(* IEC 61131-3 sources: AXOpen/src/data/tests/AXOpen.Repository.Integration.Tests_L4/ax/src, 6 files *)

(* ---- AxoDataExchange.st ---- *)
USING AXOpen.Core;
USING AXOpen;
using AXOpen.Data;

NAMESPACE Exchange_Test_L4

    {S7.extern=ReadWrite}
    CLASS PUBLIC Context EXTENDS AXOpen.Core.AxoContext
        VAR PUBLIC

            DataManager  : ProcessManager;

        END_VAR

        METHOD OVERRIDE Main

        END_METHOD
    END_CLASS

    {S7.extern=ReadWrite}
    CLASS PUBLIC ProcessManager EXTENDS AXOpen.Data.AxoDataExchange
        VAR PUBLIC
            {#ix-generic:TOnline}
            {#ix-generic:TPlain as POCO}
            {#ix-attr:[AXOpen.Data.AxoDataEntityAttribute]}
            Set : ProcessData;
        END_VAR
    END_CLASS

    {S7.extern=ReadWrite}
    CLASS PUBLIC ProcessData EXTENDS AXOpen.Data.AxoDataEntity
        VAR PUBLIC
            vString : STRING;
            vInt : INT;
            vBool : BOOL;
            NestObj : NestedObject;
        END_VAR
    END_CLASS

    {S7.extern=ReadWrite}
    CLASS PUBLIC NestedObject
        VAR PUBLIC
            vString : STRING;
            vInt : INT;
            vBool : BOOL;
        END_VAR
    END_CLASS

END_NAMESPACE

(* ---- AxoDataExchange_Test_L4.st ---- *)
USING AXOpen.Core;
USING AXOpen;
using AXOpen.Data;

NAMESPACE DataFramentsExchange_Test_L4

    //<ContextDeclaration>
    {S7.extern=ReadWrite}
    CLASS PUBLIC Context EXTENDS AXOpen.Core.AxoContext
        VAR PUBLIC

            DataManager  : AxoProcessDataManager_Test_L4;

        END_VAR

        METHOD OVERRIDE Main

        END_METHOD
    END_CLASS
    //</ContextDeclaration>

    //<AxoProcessDataManagerDeclaration>
    {S7.extern=ReadWrite}
    CLASS PUBLIC AxoProcessDataManager_Test_L4 EXTENDS AXOpen.Data.AxoDataExchange
        VAR PUBLIC
            {#ix-generic:TOnline}
            {#ix-generic:TPlain as POCO}
            {#ix-attr:[AXOpen.Data.AxoDataEntityAttribute]}
            Set : AxoProcessData_Test_L4; // <- Manager will operate on this member.
        END_VAR
    END_CLASS
    //</AxoProcessDataManagerDeclaration>

    //<AxoProcessDataDeclaration>
    {S7.extern=ReadWrite}
    CLASS PUBLIC AxoProcessData_Test_L4 EXTENDS AXOpen.Data.AxoDataEntity
        VAR PUBLIC
            vString : STRING;
            vInt : INT;
            vBool : BOOL;
            NestObj : NestingData;
        END_VAR
    END_CLASS
    //</AxoProcessDataDeclaration>

    {S7.extern=ReadWrite}
    CLASS PUBLIC NestingData
        VAR PUBLIC
            vString : STRING;
            vInt : INT;
            vBool : BOOL;
        END_VAR
    END_CLASS

END_NAMESPACE

(* ---- AxoDataFragmentExchange.st ---- *)
USING AXOpen.Core;
USING AXOpen.Data;

NAMESPACE FragmentExchange_Test_L4

    {S7.extern=ReadWrite}
    CLASS PUBLIC Context EXTENDS AXOpen.Core.AxoContext
        VAR PUBLIC
            DataManager  : FragmentProcessDataManager;
        END_VAR

        METHOD OVERRIDE Main

        END_METHOD
    END_CLASS

    {S7.extern=ReadWrite}
    CLASS PUBLIC FragmentProcessDataManager
        EXTENDS AXOpen.Data.AxoDataFragmentExchange
        VAR PUBLIC
            {#ix-attr:[AXOpen.Data.AxoDataFragmentAttribute]}
            Header : HeaderManager;

            {#ix-attr:[AXOpen.Data.AxoDataFragmentAttribute]}
            St1 : StationManager;

        END_VAR
    END_CLASS

    {S7.extern=ReadWrite}
    CLASS PUBLIC HeaderManager
        EXTENDS AXOpen.Data.AxoDataExchange
        VAR PUBLIC
            {#ix-generic:TOnline}
            {#ix-generic:TPlain as POCO}
            {#ix-attr:[AXOpen.Data.AxoDataEntityAttribute]}
            {#ix-attr:[Container(Layout.Stack)]}
            {#ix-set:AttributeName = "Shared Header"}
            Set : HeaderData;
        END_VAR
    END_CLASS

    {S7.extern=ReadWrite}
    CLASS PUBLIC HeaderData
        EXTENDS AXOpen.Data.AxoDataEntity
        VAR PUBLIC
            vString : STRING;
            vInt : INT;
            vBool : BOOL;
        END_VAR
    END_CLASS

    {S7.extern=ReadWrite}
    CLASS PUBLIC StationManager
        EXTENDS AXOpen.Data.AxoDataExchange
        VAR PUBLIC
            {#ix-generic:TOnline}
            {#ix-generic:TPlain as POCO}
            {#ix-attr:[AXOpen.Data.AxoDataEntityAttribute]}
            {#ix-attr:[Container(Layout.Stack)]}
            {#ix-set:AttributeName = "Station"}
            Set : StationData;
        END_VAR
    END_CLASS

    {S7.extern=ReadWrite}
    CLASS PUBLIC StationData EXTENDS AXOpen.Data.AxoDataEntity
        VAR PUBLIC
            vString : STRING;
            vInt : INT;
            vBool : BOOL;
            NestObj : NestedObject;
        END_VAR
    END_CLASS

    {S7.extern=ReadWrite}
    CLASS PUBLIC NestedObject
        VAR PUBLIC
            vString : STRING;
            vInt : INT;
            vBool : BOOL;
        END_VAR
    END_CLASS

END_NAMESPACE

(* ---- AxoDataFragmentExchange_Test_L4.st ---- *)
USING AXOpen.Core;
USING AXOpen.Data;

NAMESPACE AxoDataFragmentExchange_Test_L4

    //<ContextDeclaration>
    {S7.extern=ReadWrite}
    CLASS PUBLIC Context EXTENDS AXOpen.Core.AxoContext
        VAR PUBLIC

            DataManager  : AxoProcessDataManager_Test_L4;

        END_VAR

        METHOD OVERRIDE Main

        END_METHOD
    END_CLASS

    {S7.extern=ReadWrite}
    CLASS PUBLIC AxoProcessDataManager_Test_L4
        EXTENDS AXOpen.Data.AxoDataFragmentExchange
        VAR PUBLIC
            {#ix-attr:[AXOpen.Data.AxoDataFragmentAttribute]}
            Header : SharedDataHeaderManager_Test_L4;

            {#ix-attr:[AXOpen.Data.AxoDataFragmentAttribute]}
            St1 : StationProcessDataManager_Test_L4;

        END_VAR
    END_CLASS

    {S7.extern=ReadWrite}
    CLASS PUBLIC SharedDataHeaderManager_Test_L4
        EXTENDS AXOpen.Data.AxoDataExchange
        VAR PUBLIC
            {#ix-generic:TOnline}
            {#ix-generic:TPlain as POCO}
            {#ix-attr:[AXOpen.Data.AxoDataEntityAttribute]}
            {#ix-attr:[Container(Layout.Stack)]}
            {#ix-set:AttributeName = "Shared Header"}
            Set : SharedDataHeaderData_Test_L4;
        END_VAR
    END_CLASS

    {S7.extern=ReadWrite}
    CLASS PUBLIC SharedDataHeaderData_Test_L4
        EXTENDS AXOpen.Data.AxoDataEntity
        VAR PUBLIC
            SomeString : STRING;
            SomeInt : INT;
            SomeBool : BOOL;
        END_VAR
    END_CLASS

    {S7.extern=ReadWrite}
    CLASS PUBLIC StationProcessDataManager_Test_L4
        EXTENDS AXOpen.Data.AxoDataExchange
        VAR PUBLIC
            {#ix-generic:TOnline}
            {#ix-generic:TPlain as POCO}
            {#ix-attr:[AXOpen.Data.AxoDataEntityAttribute]}
            {#ix-attr:[Container(Layout.Stack)]}
            {#ix-set:AttributeName = "Station"}
            Set : StationData_Test_L4;
        END_VAR
    END_CLASS

    {S7.extern=ReadWrite}
    CLASS PUBLIC StationData_Test_L4 EXTENDS AXOpen.Data.AxoDataEntity
        VAR PUBLIC
            vString : STRING;
            vInt : INT;
            vBool : BOOL;
            NestObj : NestingData;
        END_VAR
    END_CLASS

    {S7.extern=ReadWrite}
    CLASS PUBLIC NestingData
        VAR PUBLIC
            vString : STRING;
            vInt : INT;
            vBool : BOOL;
        END_VAR
    END_CLASS

END_NAMESPACE

(* ---- configuration.st ---- *)
USING AXOpen.Data;
CONFIGURATION MyConfiguration
    TASK Main(Interval := T#10ms, Priority := 1);
    PROGRAM P1 WITH Main: MyProgram;

    VAR_GLOBAL
        {S7.extern=ReadWrite}
        AxoDataExchangeContext_Test_L4 : DataExchange_Test_L4.Context;
        {S7.extern=ReadWrite}
        AxoDataFragmentsExchangeContext_Test_L4 : DataFramentsExchange_Test_L4.Context;
    END_VAR
END_CONFIGURATION

(* ---- program.st ---- *)
PROGRAM MyProgram
    VAR_EXTERNAL
        AxoDataExchangeContext : AxoDataExchangeExample.Context;
        AxoDataFragmentsExchangeContext : AxoDataFramentsExchangeExample.Context;
    END_VAR

    AxoDataExchangeContext.Run();
    AxoDataFragmentsExchangeContext.Run();

END_PROGRAM
